// TIA Portal V20 export
// export: Created 2025-12-01T14:57:26.3740546Z, ExportSetting None, DisplayName Totally Integrated Automation Portal, DisplayVersion V20 Update 3, DisplayName TIA Portal Openness, DisplayVersion V20 Update 3, DisplayName TIA Portal Version Control Interface, DisplayVersion V20 Update 3, DisplayName STEP 7 Professional, DisplayVersion V20 Update 3, DisplayName STEP 7 Safety, DisplayVersion V20 Update 2, DisplayName WinCC Basic/Comfort/Advanced, DisplayVersion V20 Update 3, DisplayName WinCC Professional, DisplayVersion V20 Update 3, DisplayName WinCC Unified, DisplayVersion V20 Update 3
DATA_BLOCK "DB945_Datos_BWU4893"   // DB945
{ S7_Optimized_Access := 'FALSE' }
// stored: AutoNumber false
   VAR
      tarjeta : Array[1..100] of Struct
         consigna_1 : SInt;
         consigna_2 : SInt;
         consigna_3 : SInt;
         consigna_4 : SInt;
         rampa_1 : Real;
         rampa_2 : Real;
         rampa_3 : Real;
         rampa_4 : Real;
         Consigna_convertida_1 : SInt;
         Consigna_convertida_2 : SInt;
         Consigna_convertida_3 : SInt;
         Consigna_convertida_4 : SInt;
         Rampa_convertida_1 : USInt;
         Rampa_convertida_2 : USInt;
         Rampa_convertida_3 : USInt;
         Rampa_convertida_4 : USInt;
      END_STRUCT;
   END_VAR
BEGIN
   tarjeta[1].consigna_1 := -30;
   tarjeta[12].consigna_1 := -60;
   tarjeta[12].consigna_2 := 60;
   tarjeta[12].consigna_3 := -60;
   tarjeta[12].consigna_4 := 60;
   tarjeta[12].rampa_1 := 0.0;
   tarjeta[12].rampa_2 := 0.0;
   tarjeta[12].rampa_3 := 0.0;
END_DATA_BLOCK
